// Quiet by default. Eighty Info events bury the two Errors, and the counts are

// already available through I_TestRunStatus for anyone who wants them.

//

// The Verbose severity exists for narration and is filtered out of most views

// anyway - but not raising the event at all is cheaper still.
FUNCTION_BLOCK TEST_EventReporterIsQuietAboutPasses IMPLEMENTS I_Test
VAR
	Sink		  : TestEventReporter;
	ExpectedCount : UDINT;
	ActualCount	  : UDINT;
END_VAR

METHOD Run : BOOL
VAR_INPUT
	Enable : BOOL;
	Test   : I_TestAssertions;
END_VAR
Sink.TestFinished(SuiteLabel	:= 'suite',
				  TestLabel		:= 'a pass',
				  Location		:= '',
				  Status		:= E_TestStatus.Passed,
				  Kind			:= E_FailureKind.None,
				  Summary		:= '',
				  ElapsedTime	:= 0.0,
				  ElapsedCycles := 1,
				  Assertions	:= 1);

ExpectedCount := 0;
ActualCount	  := Sink.EventsSent;
Test.AssertEqual(ExpectedCount, ActualCount, 'nothing was raised');
Sink.SetVerbosity(TRUE);
Sink.TestFinished(SuiteLabel	:= 'suite',
				  TestLabel		:= 'a pass',
				  Location		:= '',
				  Status		:= E_TestStatus.Passed,
				  Kind			:= E_FailureKind.None,
				  Summary		:= '',
				  ElapsedTime	:= 0.0,
				  ElapsedCycles := 1,
				  Assertions	:= 1);

ExpectedCount := 1;
ActualCount	  := Sink.EventsSent;
Test.AssertEqual(ExpectedCount, ActualCount, 'and narration turns it on');
ExpectedCount := 0;
ActualCount	  := Sink.FailedSends;
Test.AssertEqual(ExpectedCount, ActualCount, 'the Verbose event was accepted too');
Run := TRUE;
END_METHOD

END_FUNCTION_BLOCK

(* stored: Version 1.1.0.1, ProductVersion 3.1.4026.18
   POU TEST_EventReporterIsQuietAboutPasses: Id {3f0211d5-c37a-420d-99cf-caa3c6823bd9}, SpecialFunc None
   Folder I_Test: Id {011b9096-3792-4f75-97e6-3852e1456336}
   Method Run: Id {41add4f2-4512-4d8b-8cdf-f8a051e279cf} *)
